PROGRAM PRG_Test
VAR
	convertFunctionsTest : ConvertFunctionsTest;
	periodicTriggerTest : PeriodicTriggerTest;
END_VAR

TcUnit.RUN();

END_PROGRAM

(* stored: Version 1.1.0.1, ProductVersion 3.1.4024.15
   POU PRG_Test: Id {c6742641-04bf-0196-0ddd-a724414d1ebe}, SpecialFunc None *)
